// TIA Portal V18 export
FUNCTION_BLOCK "FB21-Flush A"   // FB21, LAD
{ S7_Optimized_Access := 'TRUE' }
VERSION : 0.1
// stored: AutoNumber false, IsIECCheckEnabled false, IsRetainMemResEnabled false, MemoryReserve 100, SetENOAutomatically false, UDAEnableTagReadback false
   VAR_INPUT
      "Time" : DInt;
      "Pump ON delay" : DInt;
      "Pump OFF delay" : DInt;
   END_VAR
   VAR_OUTPUT
      "dispensing Time PV" : Int;
   END_VAR
   VAR_IN_OUT
      start : Bool;
      "Stop Flush" : Bool;
      "Flush  Running" : Bool;
      "Flush completed" : Bool;
      "ON Gear Pump" : Bool;
   END_VAR
   VAR
      "dispensing time done" : Bool;
      "dispensing time in sec" : DInt;
      "timer input" : DInt;
      IEC_Timer_0_Instance { S7_SetPoint := 'True'} : TON_TIME;
      IEC_Timer_0_Instance_1 { S7_SetPoint := 'True'} : TON_TIME;
      IEC_Timer_0_Instance_2 { S7_SetPoint := 'True'} : TON_TIME;
      IEC_Timer_0_Instance_3 { S7_SetPoint := 'True'} : TON_TIME;
   END_VAR
   VAR_TEMP   // added for the SCL form of the ladder/FBD networks
      _w1 : Bool;
   END_VAR
BEGIN

REGION Network 1
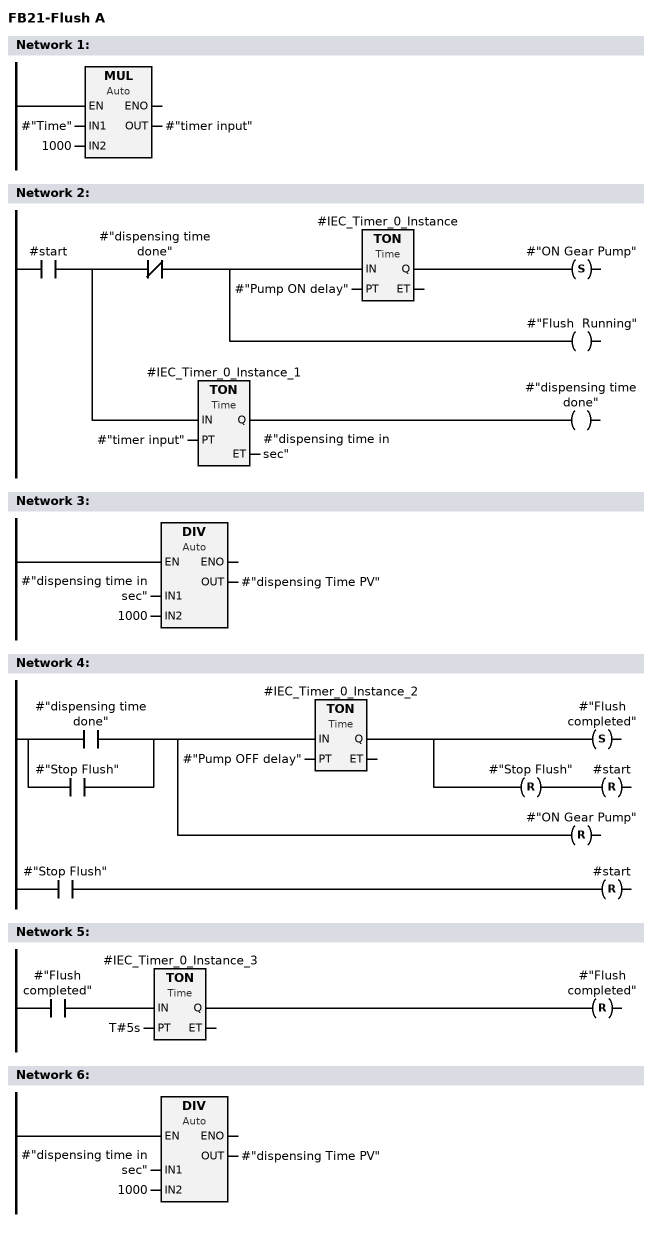
   RUNG wire#powerrail
      Mul(in1 := #"Time", in2 := 1000, out => #"timer input")
   END_RUNG
   // the same network as SCL:
   #"timer input" := #"Time" * 1000;
END_REGION

REGION Network 2
   RUNG wire#powerrail
      Contact( #start )
      wire#w1
      I_Contact( #"dispensing time done" )
      wire#w2
      { S7_Templates := "time_type := Time" } #IEC_Timer_0_Instance.TON(pt := #"Pump ON delay", et =>)
      S_Coil( #"ON Gear Pump" )
   END_RUNG
   RUNG wire#w2
      Coil( #"Flush  Running" )
   END_RUNG
   RUNG wire#w1
      { S7_Templates := "time_type := Time" } #IEC_Timer_0_Instance_1.TON(pt := #"timer input", et => #"dispensing time in sec")
      Coil( #"dispensing time done" )
   END_RUNG
   // the same network as SCL:
   #_w1 := #start AND NOT #"dispensing time done";
   #IEC_Timer_0_Instance(IN := #_w1, PT := #"Pump ON delay");   // TON
   IF #IEC_Timer_0_Instance.Q THEN #"ON Gear Pump" := TRUE; END_IF;
   #"Flush  Running" := #_w1;
   #IEC_Timer_0_Instance_1(IN := #start, PT := #"timer input", ET => #"dispensing time in sec");   // TON
   #"dispensing time done" := #IEC_Timer_0_Instance_1.Q;
END_REGION

REGION Network 3
   RUNG wire#powerrail
      Div(in1 := #"dispensing time in sec", in2 := 1000, out => #"dispensing Time PV")
   END_RUNG
   // the same network as SCL:
   #"dispensing Time PV" := #"dispensing time in sec" / 1000;
END_REGION

REGION Network 4
   RUNG wire#powerrail
      Contact( #"dispensing time done" )
      wire#w1
      { S7_Templates := "time_type := Time" } #IEC_Timer_0_Instance_2.TON(pt := #"Pump OFF delay", et =>)
      wire#w2
      S_Coil( #"Flush completed" )
   END_RUNG
   RUNG wire#powerrail
      Contact( #"Stop Flush" )
   END_RUNG wire#w1
   RUNG wire#w2
      R_Coil( #"Stop Flush" )
      R_Coil( #start )
   END_RUNG
   RUNG wire#w1
      R_Coil( #"ON Gear Pump" )
   END_RUNG
   RUNG wire#powerrail
      Contact( #"Stop Flush" )
      R_Coil( #start )
   END_RUNG
   // the same network as SCL:
   #_w1 := #"dispensing time done" OR #"Stop Flush";
   #IEC_Timer_0_Instance_2(IN := #_w1, PT := #"Pump OFF delay");   // TON
   IF #IEC_Timer_0_Instance_2.Q THEN
       #"Flush completed" := TRUE;
       #"Stop Flush" := FALSE;
       #start := FALSE;
   END_IF;
   IF #_w1 THEN #"ON Gear Pump" := FALSE; END_IF;
   IF #"Stop Flush" THEN #start := FALSE; END_IF;
END_REGION

REGION Network 5
   RUNG wire#powerrail
      Contact( #"Flush completed" )
      { S7_Templates := "time_type := Time" } #IEC_Timer_0_Instance_3.TON(pt := T#5s, et =>)
      R_Coil( #"Flush completed" )
   END_RUNG
   // the same network as SCL:
   #IEC_Timer_0_Instance_3(IN := #"Flush completed", PT := T#5s);   // TON
   IF #IEC_Timer_0_Instance_3.Q THEN #"Flush completed" := FALSE; END_IF;
END_REGION

REGION Network 6
   RUNG wire#powerrail
      Div(in1 := #"dispensing time in sec", in2 := 1000, out => #"dispensing Time PV")
   END_RUNG
   // the same network as SCL:
   #"dispensing Time PV" := #"dispensing time in sec" / 1000;
END_REGION
END_FUNCTION_BLOCK
